// TIA Portal V16 export
// export: Created 2023-08-28T09:37:32.8908657Z, ExportSetting WithDefaults, DisplayName Totally Integrated Automation Portal, DisplayVersion V16 Update 6, DisplayName TIA Portal Version Control Interface, DisplayVersion V16 Update 2, DisplayName TIA Portal Openness, DisplayVersion V16 Update 6, DisplayName STEP 7 Professional, DisplayVersion V16 Update 6, DisplayName STEP 7 Safety, DisplayVersion V16, DisplayName WinCC Advanced, DisplayVersion V16 Update 6
FUNCTION_BLOCK "01_E_PID_Reset"   // FB6, LAD
TITLE = Reset regulator PID
{ S7_Optimized_Access := 'TRUE' }
AUTHOR : rtecmer
VERSION : 0.1
// Funkcja przeprowadza reset regulatora PID gdy utraci tryb automat czyli 3
// stored: AutoNumber true, IsIECCheckEnabled false, IsRetainMemResEnabled false, MemoryReserve 100, SetENOAutomatically false, UDAEnableTagReadback false
BEGIN

REGION Network 2: Histereza reset PID
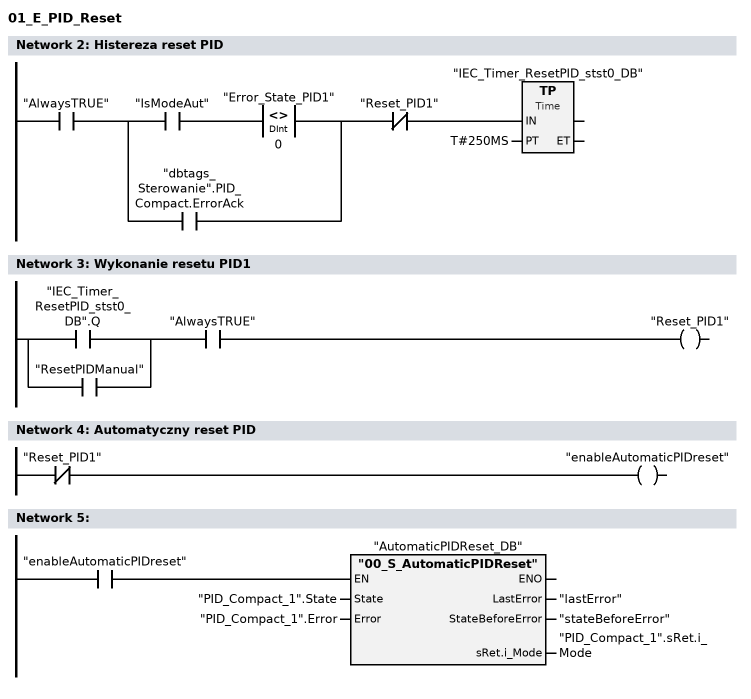
   RUNG wire#powerrail
      Contact( "AlwaysTRUE" )
      wire#w1
      Contact( "IsModeAut" )
      { S7_Templates := "SrcType := DInt" } NE_Contact(in1 := "Error_State_PID1", in2 := 0)
      wire#w2
      I_Contact( "Reset_PID1" )
      { S7_Templates := "time_type := Time" } "IEC_Timer_ResetPID_stst0_DB".TP(pt := T#250MS, et =>)
   END_RUNG
   RUNG wire#w1
      Contact( "dbtags_Sterowanie".PID_Compact.ErrorAck )
   END_RUNG wire#w2
   // the same network as SCL:
   "IEC_Timer_ResetPID_stst0_DB".TP(IN := "AlwaysTRUE" AND (("IsModeAut" AND ("Error_State_PID1" <> 0)) OR "dbtags_Sterowanie".PID_Compact.ErrorAck) AND NOT "Reset_PID1",
                           PT := T#250MS);
END_REGION

REGION Network 3: Wykonanie resetu PID1
   RUNG wire#powerrail
      Contact( "IEC_Timer_ResetPID_stst0_DB".Q )
      wire#w1
      Contact( "AlwaysTRUE" )
      Coil( "Reset_PID1" )
   END_RUNG
   RUNG wire#powerrail
      Contact( "ResetPIDManual" )
   END_RUNG wire#w1
   // the same network as SCL:
   "Reset_PID1" := ("IEC_Timer_ResetPID_stst0_DB".Q OR "ResetPIDManual") AND "AlwaysTRUE";
END_REGION

REGION Network 4: Automatyczny reset PID
   RUNG wire#powerrail
      I_Contact( "Reset_PID1" )
      Coil( "enableAutomaticPIDreset" )
   END_RUNG
   // the same network as SCL:
   "enableAutomaticPIDreset" := NOT "Reset_PID1";
END_REGION

REGION Network 5
   RUNG wire#powerrail
      Contact( "enableAutomaticPIDreset" )
      "AutomaticPIDReset_DB"(State := "PID_Compact_1".State, Error := "PID_Compact_1".Error, LastError => "lastError", StateBeforeError => "stateBeforeError", "sRet.i_Mode" => "PID_Compact_1".sRet.i_Mode)
   END_RUNG
   // the same network as SCL:
   IF "enableAutomaticPIDreset" THEN
       "AutomaticPIDReset_DB"(State := "PID_Compact_1".State,   // "00_S_AutomaticPIDReset"
                              Error := "PID_Compact_1".Error,
                              LastError => "lastError",
                              StateBeforeError => "stateBeforeError",
                              "sRet.i_Mode" => "PID_Compact_1".sRet.i_Mode);
   END_IF;
END_REGION
END_FUNCTION_BLOCK
